/// configuration data that is used during boot to configure the Units equipment
TYPE MachineDataConfig :
STRUCT
  Simulated : BOOL;
END_STRUCT
END_TYPE

(* stored: Version 1.1.0.1
   DUT MachineDataConfig: Id {ebe0a4b9-10c7-405c-a589-8dba88590acb} *)
